DATA_BLOCK "InstCounter"
{ S7_Optimized_Access := 'TRUE' }
VERSION : 0.1
NON_RETAIN
"Counter"

BEGIN

END_DATA_BLOCK

